// LS Electric XG5000 project: FDASFADS
// PLC NewPLC
// module base 0 slot 0: 입출력 모듈:XBC-DR32H (DC 24V 입력/RELAY 출력, 32점)
// module base 0 slot 1: 위치결정 모듈:XBF-PD02A (라인드라이버, 2축)
// module base 0 slot 2: 출력 모듈:XBE-TN/TP16A (TR 출력, 16점)

PROGRAM NewProgram (task: 스캔 프로그램)

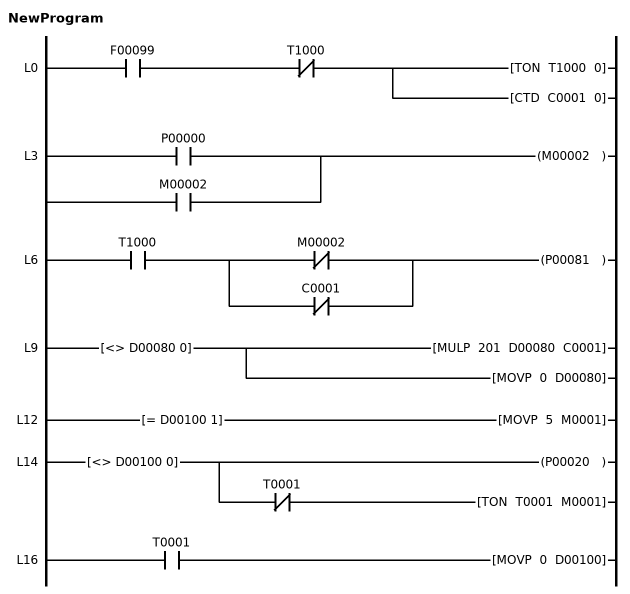
; L0
LOAD      F00099
AND NOT   T1000
TON       T1000 0
CTD       C0001 0
; L3
LOAD      P00000
OR        M00002
OUT       M00002
; L6
LOAD      T1000
LOAD NOT  M00002
OR NOT    C0001
AND LOAD
OUT       P00081
; L9
LOAD<>    D00080 0
MULP      201 D00080 C0001
MOVP      0 D00080
; L12
LOAD=     D00100 1
MOVP      5 M0001
; L14
LOAD<>    D00100 0
OUT       P00020
AND NOT   T0001
TON       T0001 M0001
; L16
LOAD      T0001
MOVP      0 D00100